{attribute 'qualified_only'}
{attribute 'strict'}
TYPE E_Hoymiles_PV_Error :
(
	eNoError := 0,
	eModbusTCPError := 1,
	eHoymilesError := 2,
	eHoymilesTooBigValueReceived := 3
);
END_TYPE

(* stored: Version 1.1.0.1, ProductVersion 3.1.4024.11
   DUT E_Hoymiles_PV_Error: Id {867d4510-bc80-4284-87c3-6b1ff591a0d3} *)
